(* PLC project Unnamed, Unknown Unnamed 1 *)
(* stored: creationDateTime 2026-05-04T21:58:54, modificationDateTime 2026-05-04T21:58:54 *)

(* simple boolean *)
PROGRAM main
  VAR
    SwitchA : BOOL := TRUE;
    SwitchB : BOOL := FALSE;
    Light : BOOL;
  END_VAR

            Light := SwitchA AND NOT SwitchB;
          
END_PROGRAM

CONFIGURATION Config0
  RESOURCE Res0 ON PLC
    TASK task0(INTERVAL := T#20ms, PRIORITY := 1);
    PROGRAM instance0 WITH task0 : main;
  END_RESOURCE
END_CONFIGURATION
